FUNCTION_BLOCK FB_ExampleDevice EXTENDS FB_Device
VAR_INPUT
END_VAR
VAR_OUTPUT
END_VAR
VAR
END_VAR

END_FUNCTION_BLOCK

(* stored: Version 1.1.0.1, ProductVersion 3.1.4024.11
   POU FB_ExampleDevice: Id {6a02f6dc-2c7b-486a-91fb-759c6a7468c4}, SpecialFunc None *)
